PROGRAM MAIN
VAR
	Controller : ConveyorController;
END_VAR

Controller();

END_PROGRAM

(* stored: Version 1.1.0.1, ProductVersion 3.1.4024.12
   POU MAIN: Id {9125b42d-76e9-46bb-903f-a0fc0ca68154}, SpecialFunc None *)
